FUNCTION Limiter : BOOL
VAR_INPUT
	fInput : REAL;
	fUpperLimit : REAL;
	fLowerLimit : REAL;
END_VAR
VAR
END_VAR

IF fInput <= fUpperLimit AND fInput >= fLowerLimit THEN
	Limiter := TRUE;
ELSE
	Limiter := FALSE;		
END_IF

END_FUNCTION

(* stored: Version 1.1.0.1, ProductVersion 3.1.4024.10
   POU Limiter: Id {c83406b6-8449-4b56-9fd0-e0580ed56c07}, SpecialFunc None *)
